% RSLogix 500 project P5_BAK012.RSS, saved by version 12.00.00.00 %
PROJECT "UNTITLED"    % processor: Bul.1763 MicroLogix 1100 Series B %

PROGRAM FILES
  LAD 2   7 rungs

DATA FILES
  O0 OUTPUT  4 elements
  I1 INPUT  6 elements
  S2 STATUS  66 elements
  B3 BINARY  1 elements
  T4 TIMER  3 elements
  C5 COUNTER  1 elements
  R6 CONTROL  1 elements
  N7 INTEGER  1 elements
  F8 FLOAT  1 elements

LADDER 2
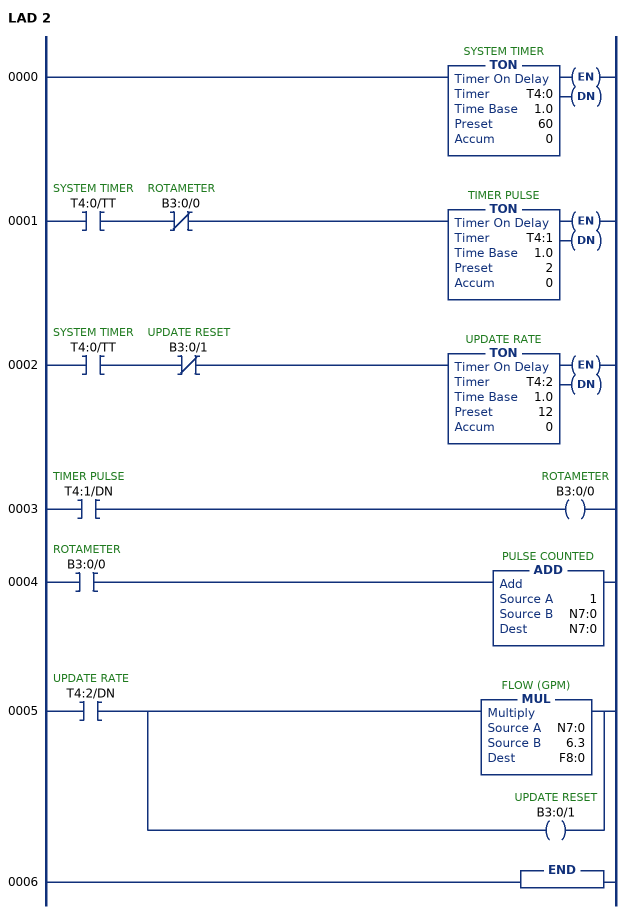
% Rung: 0 %
SOR TON T4:0 1.0 60 0 EOR
%   T4:0  "SYSTEM TIMER" %
% Rung: 1 %
SOR XIC T4:0/TT XIO B3:0/0 TON T4:1 1.0 2 0 EOR
%   T4:0  "SYSTEM TIMER" %
%   B3:0/0  "ROTAMETER" %
%   T4:1  "TIMER PULSE" %
% Rung: 2 %
SOR XIC T4:0/TT XIO B3:0/1 TON T4:2 1.0 12 0 EOR
%   T4:0  "SYSTEM TIMER" %
%   B3:0/1  "UPDATE RESET" %
%   T4:2  "UPDATE RATE" %
% Rung: 3 %
SOR XIC T4:1/DN OTE B3:0/0 EOR
%   T4:1/DN  "TIMER PULSE" %
%   B3:0/0  "ROTAMETER" %
% Rung: 4 %
SOR XIC B3:0/0 ADD 1 N7:0 N7:0 EOR
%   B3:0/0  "ROTAMETER" %
%   N7:0  "PULSE COUNTED" %
% Rung: 5 %
SOR XIC T4:2/DN BST MUL N7:0 6.3 F8:0 NXB OTE B3:0/1 BND EOR
%   T4:2  "UPDATE RATE" %
%   N7:0  "PULSE COUNTED" %
%   F8:0  "FLOW (GPM)" %
%   B3:0/1  "UPDATE RESET" %
% Rung: 6 %
SOR END EOR

DATA TABLE (non-zero values as saved)
DATA T4
% .PRE .ACC %
% T4:0 % 60 0
% T4:1 % 2 0
% T4:2 % 12 0
